Fanuc KAREL source: kd00007.KL

-- PROVISIONAL review KL for V940-1; original PC SHA256 4f183baac68cbb68badfbb75bc4914b4f8f11ca3e0eadca00d8e97da65590a0a
-- Incomplete behavior may be omitted. Consult companion uncertainty JSON. Do not deploy.
PROGRAM KD00007
%NOLOCKGROUP
-- UNRESOLVED_DECL I type=020010
-- UNRESOLVED_DECL J type=020010
-- UNRESOLVED_DECL B type=020012
-- UNRESOLVED_DECL R type=020011
-- UNRESOLVED_DECL S type=021f50
BEGIN
  -- V9_ZERO_TABLE_METADATA_HINT layout=0001; no indexed target words; source/name/runtime held
  -- UNRESOLVED_PC offsets 5-12; opcodes 9D,23
  -- UNRESOLVED_PC offsets 17-21; opcodes 7F
END KD00007
